Staubli VAL3: onExit.pgx

program onExit(bool x_bSave (dimensions=1))
  local num i
begin
  // save the saveData module
  if x_bSave
    if saveData:libSave()!=0
      delay(0.5)
      i=saveData:libSave()
      if i!=0
        popUpMsg("libsave saveData error: "+toString("",i))
        logMsg("[KERNEL] ADVANCE:Error saving saveData "+toString("",i))
      endIf
    endIf
  endIf
  //
  call use:nullKey(nKey)
end
